# B&R Automation Studio project Machine2
Automation Studio 4.9

## Configuration Config1

### Task classes (Cpu.sw)
```
Cyclic#1:
  SPL_CalcTe <- TS_UnitTest.Samples.Tests_Program.Tests_MyCalcLib_C.SPL_CalcTest.prg
  SPL_CalcT1 <- TS_UnitTest.Samples.Tests_Program.Tests_MyCalcLib_C.SPL_CalcTest_Variants.prg
  SPL_Assert <- TS_UnitTest.Samples.Framework_Extension_With_Custom_Asserts.SPL_AssertsEx.prg
  SPL_Asser1 <- TS_UnitTest.Samples.Framework_Features.SPL_Asserts.prg
  SPL_Behavi <- TS_UnitTest.Samples.Framework_Features.SPL_Behavior.prg
  utTemplate <- TS_UnitTest.Templates.HelperTool_Supported.utTemplate_automated.prg
  utTemplat1 <- TS_UnitTest.Templates.NoToolSupport.utTemplate_manual.prg
Cyclic#4:
  Counter <- Counter.prg
Libraries: LibAssert1, AsBrStr, AsARCfg, runtime, UnitTest, sys_lib, AsIecCon, astime, UtWs, UtMgr, SPLMyCalc
```

### Hardware
```
X20CP1586 : X20CP1586 v1.10.0.0
  Connector IF2:
    ActivateDevice = 1
    Mode = Manual
    InternetAddress = 192.168.1.3
    SubnetMask = 255.255.255.0
  ConfigurationID = Machine1_X20CP1583_Config1
  FileDevice1
  FileDeviceName1 = USER
  FileDevicePath1 = USER_PATH
```

## Configuration Config_X20CP1586

CPU X20CP1586, AutomationRuntime B4.93, Build 6.3.0, Vc V4.72.6

### Task classes (Cpu.sw)
```
Cyclic#1:
  SPL_CalcTe <- TS_UnitTest.Samples.Tests_Program.Tests_MyCalcLib_C.SPL_CalcTest.prg
  SPL_CalcT1 <- TS_UnitTest.Samples.Tests_Program.Tests_MyCalcLib_C.SPL_CalcTest_Variants.prg
  SPL_Assert <- TS_UnitTest.Samples.Framework_Extension_With_Custom_Asserts.SPL_AssertsEx.prg
  SPL_Asser1 <- TS_UnitTest.Samples.Framework_Features.SPL_Asserts.prg
  SPL_Behavi <- TS_UnitTest.Samples.Framework_Features.SPL_Behavior.prg
  utTemplate <- TS_UnitTest.Templates.HelperTool_Supported.utTemplate_automated.prg
  utTemplat1 <- TS_UnitTest.Templates.NoToolSupport.utTemplate_manual.prg
  ToggleOutp <- ToggleOutput.prg
Cyclic#4:
  Counter <- Counter.prg
Binaries: FWRules, TCData, udbdef, User, iomap, Role, arconfig, asfw, ashwac, sysconf, ashwd
Libraries: LibAssert1, AsBrStr, AsARCfg, runtime, UnitTest, sys_lib, AsIecCon, astime, UtWs, UtMgr, SPLMyCalc, ArProject
```

### Hardware
```
X20BM11 : X20BM11 v1.1.0.0  [X2X1 -> X20CP1586.IF6]
X20CP1586 : X20CP1586 v1.10.0.0
  Connector IF2:
    ActivateDevice = 1
    HostName = machine2
    Mode = Manual
    InternetAddress = 192.168.1.3
    SubnetMask = 255.255.255.0
  Connector IF3:
    EplHostName = machine2
    HostName = machine2
  ConfigurationID = Machine2_X20CP1586
  ConfigVersion = 1.2.3
  FileDevice1
  FileDeviceName1 = USER
  FileDevicePath1 = USER_PATH
  EthernetHostName = machine2
X20TB12 : X20TB12 v1.0.0.0
X20cDO9321 : X20cDO9321 v1.2.0.0  [SS1 -> X20TB12.SS; SL -> X20BM11.SL1]
  Supervision = off
```

### IoMap.iom - X20CP1586/IoMap.iom
```iecst
VAR_CONFIG
	::ToggleOutp:Output_1Hz AT %QX."X20cDO9321".DigitalOutput01;
	::ToggleOutp:Output_1Hz AT %QX."X20cDO9321".DigitalOutput03;
	::ToggleOutp:Output_1Hz AT %QX."X20cDO9321".DigitalOutput05;
	::ToggleOutp:Output_1Hz AT %QX."X20cDO9321".DigitalOutput07;
	::ToggleOutp:Output_1Hz AT %QX."X20cDO9321".DigitalOutput09;
	::ToggleOutp:Output_1Hz AT %QX."X20cDO9321".DigitalOutput11;
	::ToggleOutp:Output_1Hz_Inv  AT %QX."X20cDO9321".DigitalOutput02;
	::ToggleOutp:Output_1Hz_Inv  AT %QX."X20cDO9321".DigitalOutput04;
	::ToggleOutp:Output_1Hz_Inv  AT %QX."X20cDO9321".DigitalOutput06;
	::ToggleOutp:Output_1Hz_Inv  AT %QX."X20cDO9321".DigitalOutput08;
	::ToggleOutp:Output_1Hz_Inv  AT %QX."X20cDO9321".DigitalOutput10;
	::ToggleOutp:Output_1Hz_Inv  AT %QX."X20cDO9321".DigitalOutput12;
END_VAR
```

## Logical view

Binary libraries used (declarations not repeated): operator, runtime, astime, AsIecCon, AsBrStr, AsARCfg, sys_lib, ArProject


### Program Logical/Counter (ANSIC)

#### Variables.var
```iecst
VAR
	Counter : USINT;
END_VAR
```

#### Main.c
```c
#include <bur/plctypes.h>

#ifdef _DEFAULT_INCLUDES
	#include <AsDefault.h>
#endif

void _INIT ProgramInit(void)
{
	Counter = 0;
}

void _CYCLIC ProgramCyclic(void)
{
	Counter += 1;
}

void _EXIT ProgramExit(void)
{

}
```

### Program Logical/ToggleOutput

#### Variables.var
```iecst
VAR
	ActTime : UDINT;
	SetTime_1Hz : UDINT;
	Output_1Hz : BOOL;
	Output_1Hz_Inv : BOOL;
END_VAR
```

#### Main.c
```c
#include <bur/plctypes.h>

#ifdef _DEFAULT_INCLUDES
	#include <AsDefault.h>
#endif

void _INIT ProgramInit(void)
{
	Output_1Hz = 0;
}

void _CYCLIC ProgramCyclic(void)
{

	ActTime = clock_ms();

	// Toggle 1Hz
	if((ActTime-SetTime_1Hz) > 2000)
	{
		SetTime_1Hz = ActTime;
	}
	else if((ActTime-SetTime_1Hz) < 1000)
	{
		Output_1Hz = 1;
	}
	else
	{
		Output_1Hz = 0;
	}

	Output_1Hz_Inv = (Output_1Hz == 1) ? 0 : 1;
}

void _EXIT ProgramExit(void)
{

}
```

Listed in the project but not available here: Logical/Global.typ, Logical/Global.var, Logical/TS_UnitTest
